FUNCTION_BLOCK Conductor
VAR_INPUT
	vehiculo : REFERENCE TO Vehiculo(THIS^); // referencia a la clase base Vehiculo
END_VAR
VAR_OUTPUT
END_VAR
VAR
END_VAR

METHOD Mover : REAL
VAR_INPUT
	Velocidad_Deseada : REAL;
END_VAR
Mover := THIS^.vehiculo.Mover(Velocidad_Deseada);
END_METHOD

END_FUNCTION_BLOCK

(* stored: Version 1.1.0.1, ProductVersion 3.1.4024.12
   POU Conductor: Id {41072200-a029-4fd9-9fad-1cc968b7eeb8}, SpecialFunc None
   Method Mover: Id {47f83305-8310-414d-b4ea-8f95c575c437} *)
